PROGRAM auto
VAR
	ed_routine_auto: BOOL;
	redox_doser_auto_enable: BOOL;
	
	tmr_auto_pumps: TON;
	u_3112_auto_request: BOOL;
	u_3312_auto_request: BOOL;
	u_3405_auto_request: BOOL;
	u_3212_auto_request: BOOL;
	tmr_auto_pump_delay: TON;
	u_3112_running: BOOL;
	u_3112_speed_ref: INT;
	u_3112_sp: REAL;
	salt_pressure_actual: REAL;
	u_3112_ready: BOOL;
	u_3212_running: BOOL;
	u_3212_ready: BOOL;
	u_3312_ready: BOOL;
	u_3312_running: BOOL;
	u_3405_running: BOOL;
	u_3405_ready: BOOL;
	stack_power_enable: BOOL;
	nv_3110_open_request: BOOL;
	nv_3210_open_request: BOOL;
	nv_3310_open_request: BOOL;
	nv_3110_open_feedback: BOOL;
	nv_3210_open_feedback: BOOL;
	nv_3310_open_feedback: BOOL;
	nv_3110_auto_request: BOOL;
	nv_3210_auto_request: BOOL;
	nv_3310_auto_request: BOOL;

	auto_stack_power_enable: BOOL;
	AUTO_TEMP_BIT: BOOL;
END_VAR
VAR // added by the converter: edge detectors and wires of the graphical bodies
    _w1 : BOOL;
END_VAR

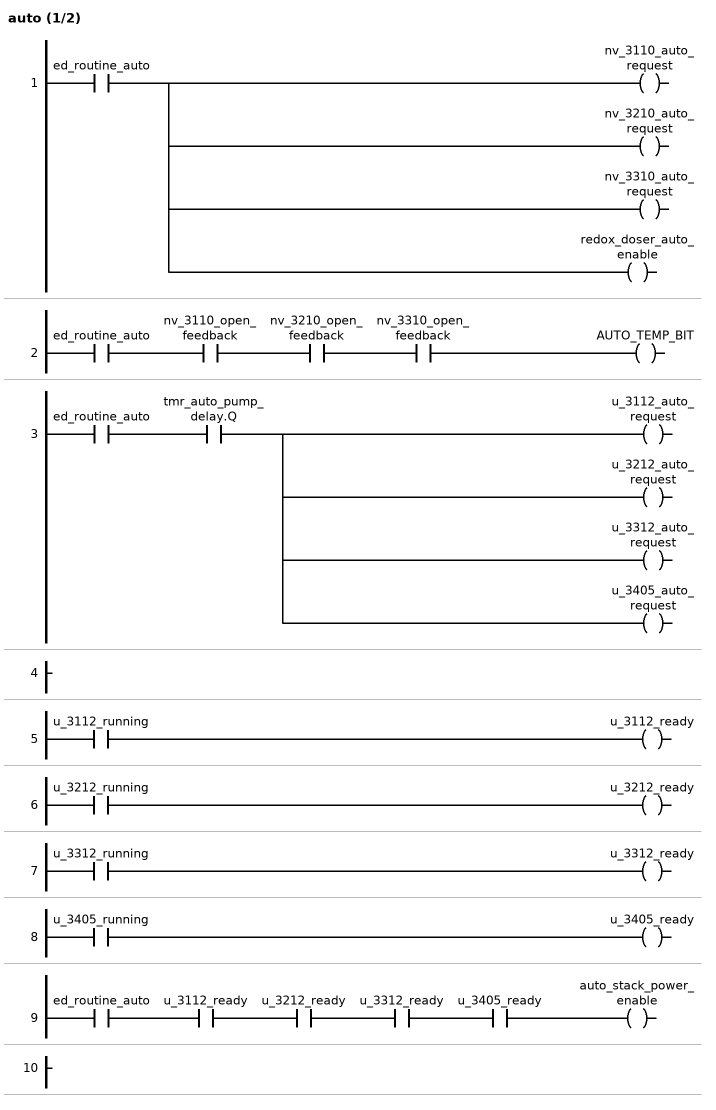
// NETWORK 1
nv_3110_auto_request := ed_routine_auto;
nv_3210_auto_request := ed_routine_auto;
nv_3310_auto_request := ed_routine_auto;
redox_doser_auto_enable := ed_routine_auto;

// NETWORK 2
AUTO_TEMP_BIT := ed_routine_auto AND nv_3110_open_feedback AND nv_3210_open_feedback AND nv_3310_open_feedback;

// NETWORK 3
_w1 := ed_routine_auto AND tmr_auto_pump_delay.Q;
u_3112_auto_request := _w1;
u_3212_auto_request := _w1;
u_3312_auto_request := _w1;
u_3405_auto_request := _w1;

// NETWORK 4

// NETWORK 5
u_3112_ready := u_3112_running;

// NETWORK 6
u_3212_ready := u_3212_running;

// NETWORK 7
u_3312_ready := u_3312_running;

// NETWORK 8
u_3405_ready := u_3405_running;

// NETWORK 9
auto_stack_power_enable := ed_routine_auto AND u_3112_ready AND u_3212_ready AND u_3312_ready AND u_3405_ready;

// NETWORK 10

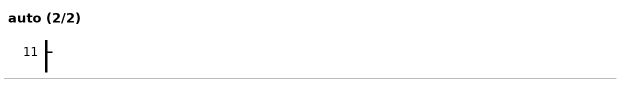
// NETWORK 11

END_PROGRAM

(* stored: Version 1.1.0.1, ProductVersion 3.1.4024.12
   POU auto: Id {3d08b1fd-a23f-437d-8121-cefd84a9c392}, SpecialFunc None *)
